FUNCTION_BLOCK FB_CraneController
VAR_INPUT
    nAisleNumber    : INT;
	iCrane          : I_Crane;
END_VAR
VAR_OUTPUT
    bBusy           : BOOL;
    bError          : BOOL;
    bPickDone       : BOOL;
    bDropDone       : BOOL;
END_VAR

VAR
    stAisleStation  : ST_Position;
    stRackTarget    : ST_Position;
    bJobPending     : BOOL;
    bIsStore        : BOOL;
    nState          : (IDLE, DISPATCHING, EXECUTING, DONE) := IDLE;
END_VAR

// Wire physical IO based on aisle
IF nAisleNumber = 1 THEN
    GVL_IO.bCrane1MotorX  := iCrane.bBusy AND GVL_IO.fCrane1PosX <> 0.0;
    GVL_IO.bCrane1MotorY  := iCrane.bBusy AND GVL_IO.fCrane1PosY <> 0.0;
END_IF

bBusy  := iCrane.bBusy;
bError := iCrane.bError;

CASE nState OF

    IDLE:
        bPickDone := FALSE;
        bDropDone := FALSE;
        IF bJobPending THEN
            nState := DISPATCHING;
        END_IF

    DISPATCHING:
        stAisleStation.fTargetX        := GVL_Config.HOME_X;
        stAisleStation.fTargetY        := GVL_Config.HOME_Y;
        stAisleStation.bIsAisleStation := TRUE;
        IF bIsStore THEN
            iCrane.M_StartJob(stPick := stAisleStation, stPlace := stRackTarget);
        ELSE
            iCrane.M_StartJob(stPick := stRackTarget, stPlace := stAisleStation);
        END_IF
        bJobPending := FALSE;
        nState      := EXECUTING;

    EXECUTING:
        IF iCrane.eState = E_CraneState.IDLE THEN
           // IF bIsStore THEN
           //     bPickDone := TRUE;
           // ELSE
			//	bDropDone := TRUE;
           // END_IF
			IF GVL_IO.bAisle1CraneStation OR GVL_IO.bAisle2CraneStation THEN
				IF nAisleNumber = 1 THEN
					GVL_IO.bCrane1pick := TRUE;
				ELSIF nAisleNumber = 2 THEN
					GVL_IO.bCrane2pick := TRUE;
				END_IF
				nState := DONE;
			END_IF
        END_IF

    DONE:
        bDropDone := FALSE;
        bPickDone := FALSE;
        nState    := IDLE;

END_CASE

IF iCrane.bError THEN
    bJobPending := FALSE;
    nState      := IDLE;
END_IF

METHOD M_AssignRetrieve : BOOL
VAR_INPUT
    stPos : ST_Position;
END_VAR
IF nState <> IDLE OR bJobPending THEN
    M_AssignRetrieve := FALSE;
    RETURN;
END_IF
stRackTarget     := stPos;
bIsStore         := FALSE;
bJobPending      := TRUE;
M_AssignRetrieve := TRUE;
END_METHOD

METHOD M_AssignStore : BOOL
VAR_INPUT
    stPos : ST_Position;
END_VAR
IF nState <> IDLE OR bJobPending THEN
    M_AssignStore := FALSE;
    RETURN;
END_IF
stRackTarget  := stPos;
bIsStore      := TRUE;
bJobPending   := TRUE;
M_AssignStore := TRUE;
END_METHOD

END_FUNCTION_BLOCK

(* stored: Version 1.1.0.1, ProductVersion 3.1.4024.16
   POU FB_CraneController: Id {a8b9c0d1-e2f3-4567-8901-234567890123}, SpecialFunc None
   Method M_AssignRetrieve: Id {dd000002-0000-0000-0000-000000000001}
   Method M_AssignStore: Id {dd000001-0000-0000-0000-000000000001} *)
